// TIA Portal V20 export
DATA_BLOCK "InstPlcDiag"   // DB34
AUTHOR : Siemens Digital Industries
FAMILY : LAF
// stored: InstanceOfName LAF_PlcDiag, InstanceOfType FB
"LAF_PlcDiag"
   // VAR_INPUT
   //    localCommon { ExternalAccessible := 'False'; ExternalVisible := 'False'; ExternalWritable := 'False'} : HW_SUBMODULE := 50;
   //    localProfinetInterface { ExternalAccessible := 'False'; ExternalVisible := 'False'; ExternalWritable := 'False'} : HW_INTERFACE := 64;
   //    firstCycle { ExternalAccessible := 'False'; ExternalVisible := 'False'; ExternalWritable := 'False'} : Bool := FALSE;
   // END_VAR
   // VAR_IN_OUT
   //    diagDataHmi : "LAF_typePlcDiag";
   // END_VAR
   // VAR
   //    statLocalCommon { ExternalAccessible := 'False'; ExternalVisible := 'False'; ExternalWritable := 'False'} : HW_SUBMODULE := 50;
   //    statLocProfinetInterface { ExternalAccessible := 'False'; ExternalVisible := 'False'; ExternalWritable := 'False'} : HW_INTERFACE := 64;
   //    instGetImData0 { ExternalAccessible := 'False'; ExternalVisible := 'False'; ExternalWritable := 'False'} : Get_IM_Data;
   //    statGetImData0ErrorSaved { ExternalAccessible := 'False'; ExternalVisible := 'False'; ExternalWritable := 'False'} : Word := 16#0000;
   //    instGetImData1 { ExternalAccessible := 'False'; ExternalVisible := 'False'; ExternalWritable := 'False'} : Get_IM_Data;
   //    statGetImData1ErrorSaved { ExternalAccessible := 'False'; ExternalVisible := 'False'; ExternalWritable := 'False'} : Word := 16#0000;
   //    instGetImData2 { ExternalAccessible := 'False'; ExternalVisible := 'False'; ExternalWritable := 'False'} : Get_IM_Data;
   //    statGetImData2ErrorSaved { ExternalAccessible := 'False'; ExternalVisible := 'False'; ExternalWritable := 'False'} : Word := 16#0000;
   //    instGetImData3 { ExternalAccessible := 'False'; ExternalVisible := 'False'; ExternalWritable := 'False'} : Get_IM_Data;
   //    statGetImData3ErroSaved { ExternalAccessible := 'False'; ExternalVisible := 'False'; ExternalWritable := 'False'} : Word := 16#0000;
   //    instReadRecord { ExternalAccessible := 'False'; ExternalVisible := 'False'; ExternalWritable := 'False'} : RDREC;
   //    statReadRecordResult { ExternalAccessible := 'False'; ExternalVisible := 'False'; ExternalWritable := 'False'} : Array[0..199] of Byte;
   //    statStartNetAddresses { ExternalAccessible := 'False'; ExternalVisible := 'False'; ExternalWritable := 'False'} : USInt := 40;
   //    statIm1PlDesiLocIdLen { ExternalAccessible := 'False'; ExternalVisible := 'False'; ExternalWritable := 'False'} : Int := 54;
   //    statRisEdgeReadAll { ExternalAccessible := 'False'; ExternalVisible := 'False'; ExternalWritable := 'False'} : Bool := FALSE;
   //    statPosPulseReadAll { ExternalAccessible := 'False'; ExternalVisible := 'False'; ExternalWritable := 'False'} : Bool := FALSE;
   //    statErrorText { ExternalAccessible := 'False'; ExternalVisible := 'False'; ExternalWritable := 'False'} : String[30] := 'Error - Not readable data';
   // END_VAR
BEGIN
   instGetImData0.LADDR := 50;
   instGetImData0.IM_TYPE := 0;
   instGetImData0.DONE := TRUE;
   instGetImData0.BUSY := FALSE;
   instGetImData0.ERROR := FALSE;
   instGetImData0.STATUS := 16#0000;
   instGetImData0.sdw_GetAttrID := 16#0000_0031;
   instGetImData0.sdw_GetAttrAID := 16#0000_0EA9;
   instGetImData0.sdi_SfcLen := 60;
   instGetImData0.sb_useGetMultiAttr := FALSE;
   instGetImData0.sui_GetMultiAttrACount := 0;
   instGetImData0.sa_GetMultiAttrPathLens[0] := 0;
   instGetImData0.sa_GetMultiAttrPaths[0..2] := 0;
   instGetImData0.sa_GetMultiAttrResultLens[0] := 0;
   instGetImData0.sa_GetMultiAttrResult := ' ';
   instGetImData0.sb_SfcValid := TRUE;
   instGetImData0.sb_SfcERROR := FALSE;
   instGetImData0.sw_SfcStatus := 16#0000;
   instGetImData0.sa_SfcData[0] := 16#00;
   instGetImData0.sa_SfcData[1] := 16#20;
   instGetImData0.sa_SfcData[2] := 16#00;
   instGetImData0.sa_SfcData[3] := 16#38;
   instGetImData0.sa_SfcData[4] := 16#01;
   instGetImData0.sa_SfcData[5..6] := 16#00;
   instGetImData0.sa_SfcData[7] := 16#2A;
   instGetImData0.sa_SfcData[8] := 16#36;
   instGetImData0.sa_SfcData[9] := 16#45;
   instGetImData0.sa_SfcData[10] := 16#53;
   instGetImData0.sa_SfcData[11] := 16#37;
   instGetImData0.sa_SfcData[12] := 16#20;
   instGetImData0.sa_SfcData[13] := 16#35;
   instGetImData0.sa_SfcData[14] := 16#31;
   instGetImData0.sa_SfcData[15] := 16#38;
   instGetImData0.sa_SfcData[16] := 16#2D;
   instGetImData0.sa_SfcData[17] := 16#33;
   instGetImData0.sa_SfcData[18] := 16#55;
   instGetImData0.sa_SfcData[19] := 16#54;
   instGetImData0.sa_SfcData[20] := 16#31;
   instGetImData0.sa_SfcData[21] := 16#30;
   instGetImData0.sa_SfcData[22] := 16#2D;
   instGetImData0.sa_SfcData[23] := 16#30;
   instGetImData0.sa_SfcData[24] := 16#41;
   instGetImData0.sa_SfcData[25] := 16#42;
   instGetImData0.sa_SfcData[26] := 16#30;
   instGetImData0.sa_SfcData[27] := 16#20;
   instGetImData0.sa_SfcData[28] := 16#53;
   instGetImData0.sa_SfcData[29] := 16#20;
   instGetImData0.sa_SfcData[30] := 16#43;
   instGetImData0.sa_SfcData[31] := 16#2D;
   instGetImData0.sa_SfcData[32] := 16#54;
   instGetImData0.sa_SfcData[33] := 16#34;
   instGetImData0.sa_SfcData[34] := 16#41;
   instGetImData0.sa_SfcData[35] := 16#30;
   instGetImData0.sa_SfcData[36] := 16#52;
   instGetImData0.sa_SfcData[37] := 16#56;
   instGetImData0.sa_SfcData[38] := 16#48;
   instGetImData0.sa_SfcData[39] := 16#4D;
   instGetImData0.sa_SfcData[40] := 16#32;
   instGetImData0.sa_SfcData[41] := 16#30;
   instGetImData0.sa_SfcData[42] := 16#32;
   instGetImData0.sa_SfcData[43] := 16#35;
   instGetImData0.sa_SfcData[44] := 16#00;
   instGetImData0.sa_SfcData[45] := 16#01;
   instGetImData0.sa_SfcData[46] := 16#56;
   instGetImData0.sa_SfcData[47] := 16#04;
   instGetImData0.sa_SfcData[48..55] := 16#00;
   instGetImData0.sa_SfcData[56..57] := 16#01;
   instGetImData0.sa_SfcData[58] := 16#00;
   instGetImData0.sa_SfcData[59] := 16#0E;
   instGetImData0.sa_SfcData[60..64] := 16#00;
   instGetImData0.sudi_arraylength := 54;
   instGetImData0.sudi_datatype := 4;
   instGetImData0.sui_imdataLen := 54;
   instGetImData0.sui_imdataLen_netto := 54;
   instGetImData0.si_index := 16;
   instGetImData0.sb_SfcLocked := FALSE;
   instGetImData0.pw_TemporaryWord := 16#000E;
   instGetImData0.pa_DataByte[0..53] := 16#00;
   instGetImData0.pa_DataChar[0..53] := ' ';
   instGetImData0.pa_TemporaryCharArray[0] := 'S';
   instGetImData0.pa_TemporaryCharArray[1] := ' ';
   instGetImData0.pa_TemporaryCharArray[2] := 'C';
   instGetImData0.pa_TemporaryCharArray[3] := '-';
   instGetImData0.pa_TemporaryCharArray[4] := 'T';
   instGetImData0.pa_TemporaryCharArray[5] := '4';
   instGetImData0.pa_TemporaryCharArray[6] := 'A';
   instGetImData0.pa_TemporaryCharArray[7] := '0';
   instGetImData0.pa_TemporaryCharArray[8] := 'R';
   instGetImData0.pa_TemporaryCharArray[9] := 'V';
   instGetImData0.pa_TemporaryCharArray[10] := 'H';
   instGetImData0.pa_TemporaryCharArray[11] := 'M';
   instGetImData0.pa_TemporaryCharArray[12] := '2';
   instGetImData0.pa_TemporaryCharArray[13] := '0';
   instGetImData0.pa_TemporaryCharArray[14] := '2';
   instGetImData0.pa_TemporaryCharArray[15] := '5';
   instGetImData0.pa_TemporaryCharArray[16] := 'A';
   instGetImData0.pa_TemporaryCharArray[17] := 'B';
   instGetImData0.pa_TemporaryCharArray[18] := '0';
   instGetImData0.pa_TemporaryCharArray[19] := ' ';
   instGetImData0.p_DataUDT.Manufacturer_ID := 42;
   instGetImData0.p_DataUDT.Order_ID := '6ES7 518-3UT10-0AB0 ';
   instGetImData0.p_DataUDT.Serial_Number := 'S C-T4A0RVHM2025';
   instGetImData0.p_DataUDT.Hardware_Revision := 1;
   instGetImData0.p_DataUDT.Software_Revision."Type" := 'V';
   instGetImData0.p_DataUDT.Software_Revision.Functional := 4;
   instGetImData0.p_DataUDT.Software_Revision.Bugfix := 0;
   instGetImData0.p_DataUDT.Software_Revision.Internal := 0;
   instGetImData0.p_DataUDT.Revision_Counter := 0;
   instGetImData0.p_DataUDT.Profile_ID := 0;
   instGetImData0.p_DataUDT.Profile_Specific_Type := 0;
   instGetImData0.p_DataUDT.IM_Version := 16#0101;
   instGetImData0.p_DataUDT.IM_Supported := 16#000E;
   instGetImData1.LADDR := 50;
   instGetImData1.IM_TYPE := 11;
   instGetImData1.DONE := TRUE;
   instGetImData1.BUSY := FALSE;
   instGetImData1.ERROR := FALSE;
   instGetImData1.STATUS := 16#0000;
   instGetImData1.sdw_GetAttrID := 16#0000_0031;
   instGetImData1.sdw_GetAttrAID := 16#0000_0000;
   instGetImData1.sdi_SfcLen := 60;
   instGetImData1.sb_useGetMultiAttr := TRUE;
   instGetImData1.sui_GetMultiAttrACount := 1;
   instGetImData1.sa_GetMultiAttrPathLens[0] := 3;
   instGetImData1.sa_GetMultiAttrPaths[0] := 49;
   instGetImData1.sa_GetMultiAttrPaths[1] := 4690;
   instGetImData1.sa_GetMultiAttrPaths[2] := 45041;
   instGetImData1.sa_GetMultiAttrResultLens[0] := 0;
   instGetImData1.sa_GetMultiAttrResult := ' ';
   instGetImData1.sb_SfcValid := TRUE;
   instGetImData1.sb_SfcERROR := FALSE;
   instGetImData1.sw_SfcStatus := 16#0000;
   instGetImData1.sa_SfcData[0] := 16#00;
   instGetImData1.sa_SfcData[1] := 16#21;
   instGetImData1.sa_SfcData[2] := 16#00;
   instGetImData1.sa_SfcData[3] := 16#38;
   instGetImData1.sa_SfcData[4] := 16#01;
   instGetImData1.sa_SfcData[5] := 16#00;
   instGetImData1.sa_SfcData[6..59] := 16#20;
   instGetImData1.sa_SfcData[60..64] := 16#00;
   instGetImData1.sudi_arraylength := 0;
   instGetImData1.sudi_datatype := 1;
   instGetImData1.sui_imdataLen := 54;
   instGetImData1.sui_imdataLen_netto := 54;
   instGetImData1.si_index := 0;
   instGetImData1.sb_SfcLocked := FALSE;
   instGetImData1.pw_TemporaryWord := 16#0000;
   instGetImData1.pa_DataByte[0..53] := 16#00;
   instGetImData1.pa_DataChar[0..53] := ' ';
   instGetImData1.pa_TemporaryCharArray[0..19] := ' ';
   instGetImData1.p_DataUDT.Manufacturer_ID := 0;
   instGetImData1.p_DataUDT.Order_ID := '';
   instGetImData1.p_DataUDT.Serial_Number := '';
   instGetImData1.p_DataUDT.Hardware_Revision := 0;
   instGetImData1.p_DataUDT.Software_Revision."Type" := ' ';
   instGetImData1.p_DataUDT.Software_Revision.Functional := 0;
   instGetImData1.p_DataUDT.Software_Revision.Bugfix := 0;
   instGetImData1.p_DataUDT.Software_Revision.Internal := 0;
   instGetImData1.p_DataUDT.Revision_Counter := 0;
   instGetImData1.p_DataUDT.Profile_ID := 0;
   instGetImData1.p_DataUDT.Profile_Specific_Type := 0;
   instGetImData1.p_DataUDT.IM_Version := 16#0000;
   instGetImData1.p_DataUDT.IM_Supported := 16#0000;
   instGetImData2.LADDR := 50;
   instGetImData2.IM_TYPE := 12;
   instGetImData2.DONE := TRUE;
   instGetImData2.BUSY := FALSE;
   instGetImData2.ERROR := FALSE;
   instGetImData2.STATUS := 16#0000;
   instGetImData2.sdw_GetAttrID := 16#0000_0031;
   instGetImData2.sdw_GetAttrAID := 16#0000_0000;
   instGetImData2.sdi_SfcLen := 22;
   instGetImData2.sb_useGetMultiAttr := TRUE;
   instGetImData2.sui_GetMultiAttrACount := 1;
   instGetImData2.sa_GetMultiAttrPathLens[0] := 3;
   instGetImData2.sa_GetMultiAttrPaths[0] := 49;
   instGetImData2.sa_GetMultiAttrPaths[1] := 4690;
   instGetImData2.sa_GetMultiAttrPaths[2] := 45042;
   instGetImData2.sa_GetMultiAttrResultLens[0] := 0;
   instGetImData2.sa_GetMultiAttrResult := ' ';
   instGetImData2.sb_SfcValid := TRUE;
   instGetImData2.sb_SfcERROR := FALSE;
   instGetImData2.sw_SfcStatus := 16#0000;
   instGetImData2.sa_SfcData[0] := 16#00;
   instGetImData2.sa_SfcData[1] := 16#22;
   instGetImData2.sa_SfcData[2] := 16#00;
   instGetImData2.sa_SfcData[3] := 16#12;
   instGetImData2.sa_SfcData[4] := 16#01;
   instGetImData2.sa_SfcData[5] := 16#00;
   instGetImData2.sa_SfcData[6] := 16#32;
   instGetImData2.sa_SfcData[7] := 16#30;
   instGetImData2.sa_SfcData[8] := 16#32;
   instGetImData2.sa_SfcData[9] := 16#35;
   instGetImData2.sa_SfcData[10] := 16#2D;
   instGetImData2.sa_SfcData[11] := 16#30;
   instGetImData2.sa_SfcData[12] := 16#32;
   instGetImData2.sa_SfcData[13] := 16#2D;
   instGetImData2.sa_SfcData[14] := 16#32;
   instGetImData2.sa_SfcData[15] := 16#34;
   instGetImData2.sa_SfcData[16] := 16#20;
   instGetImData2.sa_SfcData[17] := 16#31;
   instGetImData2.sa_SfcData[18] := 16#36;
   instGetImData2.sa_SfcData[19] := 16#3A;
   instGetImData2.sa_SfcData[20] := 16#35;
   instGetImData2.sa_SfcData[21] := 16#39;
   instGetImData2.sa_SfcData[22..64] := 16#00;
   instGetImData2.sudi_arraylength := 0;
   instGetImData2.sudi_datatype := 1;
   instGetImData2.sui_imdataLen := 16;
   instGetImData2.sui_imdataLen_netto := 16;
   instGetImData2.si_index := 0;
   instGetImData2.sb_SfcLocked := FALSE;
   instGetImData2.pw_TemporaryWord := 16#0000;
   instGetImData2.pa_DataByte[0..53] := 16#00;
   instGetImData2.pa_DataChar[0..53] := ' ';
   instGetImData2.pa_TemporaryCharArray[0..19] := ' ';
   instGetImData2.p_DataUDT.Manufacturer_ID := 0;
   instGetImData2.p_DataUDT.Order_ID := '';
   instGetImData2.p_DataUDT.Serial_Number := '';
   instGetImData2.p_DataUDT.Hardware_Revision := 0;
   instGetImData2.p_DataUDT.Software_Revision."Type" := ' ';
   instGetImData2.p_DataUDT.Software_Revision.Functional := 0;
   instGetImData2.p_DataUDT.Software_Revision.Bugfix := 0;
   instGetImData2.p_DataUDT.Software_Revision.Internal := 0;
   instGetImData2.p_DataUDT.Revision_Counter := 0;
   instGetImData2.p_DataUDT.Profile_ID := 0;
   instGetImData2.p_DataUDT.Profile_Specific_Type := 0;
   instGetImData2.p_DataUDT.IM_Version := 16#0000;
   instGetImData2.p_DataUDT.IM_Supported := 16#0000;
   instGetImData3.LADDR := 50;
   instGetImData3.IM_TYPE := 13;
   instGetImData3.DONE := TRUE;
   instGetImData3.BUSY := FALSE;
   instGetImData3.ERROR := FALSE;
   instGetImData3.STATUS := 16#0000;
   instGetImData3.sdw_GetAttrID := 16#0000_0031;
   instGetImData3.sdw_GetAttrAID := 16#0000_0000;
   instGetImData3.sdi_SfcLen := 60;
   instGetImData3.sb_useGetMultiAttr := TRUE;
   instGetImData3.sui_GetMultiAttrACount := 1;
   instGetImData3.sa_GetMultiAttrPathLens[0] := 3;
   instGetImData3.sa_GetMultiAttrPaths[0] := 49;
   instGetImData3.sa_GetMultiAttrPaths[1] := 4690;
   instGetImData3.sa_GetMultiAttrPaths[2] := 45043;
   instGetImData3.sa_GetMultiAttrResultLens[0] := 0;
   instGetImData3.sa_GetMultiAttrResult := ' ';
   instGetImData3.sb_SfcValid := TRUE;
   instGetImData3.sb_SfcERROR := FALSE;
   instGetImData3.sw_SfcStatus := 16#0000;
   instGetImData3.sa_SfcData[0] := 16#00;
   instGetImData3.sa_SfcData[1] := 16#23;
   instGetImData3.sa_SfcData[2] := 16#00;
   instGetImData3.sa_SfcData[3] := 16#38;
   instGetImData3.sa_SfcData[4] := 16#01;
   instGetImData3.sa_SfcData[5] := 16#00;
   instGetImData3.sa_SfcData[6..59] := 16#20;
   instGetImData3.sa_SfcData[60..64] := 16#00;
   instGetImData3.sudi_arraylength := 0;
   instGetImData3.sudi_datatype := 1;
   instGetImData3.sui_imdataLen := 54;
   instGetImData3.sui_imdataLen_netto := 54;
   instGetImData3.si_index := 0;
   instGetImData3.sb_SfcLocked := FALSE;
   instGetImData3.pw_TemporaryWord := 16#0000;
   instGetImData3.pa_DataByte[0..53] := 16#00;
   instGetImData3.pa_DataChar[0..53] := ' ';
   instGetImData3.pa_TemporaryCharArray[0..19] := ' ';
   instGetImData3.p_DataUDT.Manufacturer_ID := 0;
   instGetImData3.p_DataUDT.Order_ID := '';
   instGetImData3.p_DataUDT.Serial_Number := '';
   instGetImData3.p_DataUDT.Hardware_Revision := 0;
   instGetImData3.p_DataUDT.Software_Revision."Type" := ' ';
   instGetImData3.p_DataUDT.Software_Revision.Functional := 0;
   instGetImData3.p_DataUDT.Software_Revision.Bugfix := 0;
   instGetImData3.p_DataUDT.Software_Revision.Internal := 0;
   instGetImData3.p_DataUDT.Revision_Counter := 0;
   instGetImData3.p_DataUDT.Profile_ID := 0;
   instGetImData3.p_DataUDT.Profile_Specific_Type := 0;
   instGetImData3.p_DataUDT.IM_Version := 16#0000;
   instGetImData3.p_DataUDT.IM_Supported := 16#0000;
   instReadRecord.REQ := FALSE;
   instReadRecord.ID := 64;
   instReadRecord.INDEX := 32896;
   instReadRecord.MLEN := 200;
   instReadRecord.VALID := FALSE;
   instReadRecord.BUSY := FALSE;
   instReadRecord.ERROR := FALSE;
   instReadRecord.STATUS := 16#0070_0000;
   instReadRecord.LEN := 0;
   statReadRecordResult[0] := 16#02;
   statReadRecordResult[1] := 16#40;
   statReadRecordResult[2] := 16#00;
   statReadRecordResult[3] := 16#38;
   statReadRecordResult[4] := 16#01;
   statReadRecordResult[5] := 16#00;
   statReadRecordResult[6] := 16#1E;
   statReadRecordResult[7] := 16#62;
   statReadRecordResult[8] := 16#61;
   statReadRecordResult[9] := 16#30;
   statReadRecordResult[10] := 16#33;
   statReadRecordResult[11] := 16#30;
   statReadRecordResult[12] := 16#61;
   statReadRecordResult[13] := 16#7A;
   statReadRecordResult[14] := 16#73;
   statReadRecordResult[15] := 16#63;
   statReadRecordResult[16] := 16#31;
   statReadRecordResult[17] := 16#2E;
   statReadRecordResult[18] := 16#62;
   statReadRecordResult[19] := 16#61;
   statReadRecordResult[20] := 16#30;
   statReadRecordResult[21] := 16#33;
   statReadRecordResult[22] := 16#30;
   statReadRecordResult[23] := 16#61;
   statReadRecordResult[24] := 16#7A;
   statReadRecordResult[25] := 16#73;
   statReadRecordResult[26] := 16#63;
   statReadRecordResult[27] := 16#31;
   statReadRecordResult[28] := 16#78;
   statReadRecordResult[29] := 16#62;
   statReadRecordResult[30..31] := 16#78;
   statReadRecordResult[32] := 16#31;
   statReadRecordResult[33] := 16#33;
   statReadRecordResult[34] := 16#63;
   statReadRecordResult[35] := 16#33;
   statReadRecordResult[36] := 16#66;
   statReadRecordResult[37..39] := 16#00;
   statReadRecordResult[40] := 16#30;
   statReadRecordResult[41] := 16#B8;
   statReadRecordResult[42] := 16#51;
   statReadRecordResult[43] := 16#66;
   statReadRecordResult[44] := 16#CF;
   statReadRecordResult[45] := 16#66;
   statReadRecordResult[46..47] := 16#00;
   statReadRecordResult[48] := 16#C0;
   statReadRecordResult[49] := 16#A8;
   statReadRecordResult[50] := 16#C8;
   statReadRecordResult[51] := 16#33;
   statReadRecordResult[52..54] := 16#FF;
   statReadRecordResult[55] := 16#00;
   statReadRecordResult[56] := 16#C0;
   statReadRecordResult[57] := 16#A8;
   statReadRecordResult[58] := 16#C8;
   statReadRecordResult[59] := 16#33;
   statReadRecordResult[60..199] := 16#00;
END_DATA_BLOCK
